FUNCTION_BLOCK AUI_ADD_4_UNGATED (* Wie AUI_ADD_4, aber OHNE Aenderungserkennung - reicht JEDES neu berechnete Ergebnis bedingungslos weiter (fuer Verbraucher, die eine periodische Kadenz unabhaengig von Wertaenderung brauchen, z.B. Ableitungs-/Frequenzberechnungen). *)
  (* Standard: 61499-2; Description: Copyright (c) 2026 Meisterschulen am Ostbahnhof This program and the accompanying materials are made available under the terms of the Eclipse Public License 2.0 which is available at https://www.eclipse.org/legal/epl-2.0/ SPDX-License-Identifier: EPL-2.0 *)
  (* Version 1.0, 2026-08-31, Franz Höpfinger, Meisterschulen am Ostbahnhof, initial API and implementation and/or initial documentation *)
  PACKAGE adapter::iec61131::arithmetic;
  IMPORT eclipse4diac::core::GenericClassName;
  {SET_ATTRIBUTE(eclipse4diac::core::GenericClassName, 'GEN_AUI_ADD')}
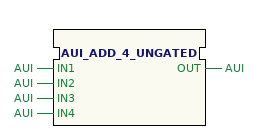
  SOCKETS
    IN1 : adapter::types::unidirectional::AUI; (* ADD input 1 *)
    IN2 : adapter::types::unidirectional::AUI; (* ADD input 2 *)
    IN3 : adapter::types::unidirectional::AUI; (* ADD input 3 *)
    IN4 : adapter::types::unidirectional::AUI; (* ADD input 4 *)
  END_SOCKETS
  PLUGS
    OUT : adapter::types::unidirectional::AUI; (* ADD result *)
  END_PLUGS
END_FUNCTION_BLOCK
